FUNCTION_BLOCK Control (* Composite Function Block Type *)
  (* Standard: 61499-2 *)
  (* Version 0.0, 2/9/2018, Sandeep Patil, nxtControl GmbH, template *)
  PACKAGE Main;
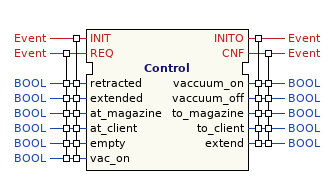
  EVENT_INPUT
    INIT WITH retracted, extended, at_magazine, at_client, empty, vac_on; (* Initialization Request *)
    REQ WITH retracted, extended, at_magazine, at_client, empty, vac_on; (* Normal Execution Request *)
  END_EVENT
  EVENT_OUTPUT
    INITO WITH vaccuum_on, vaccuum_off, to_magazine, to_client, extend; (* Initialization Confirm *)
    CNF WITH vaccuum_on, vaccuum_off, to_magazine, to_client, extend; (* Execution Confirmation *)
  END_EVENT
  VAR_INPUT
    retracted : BOOL;
    extended : BOOL;
    at_magazine : BOOL; (* Input event qualifier *)
    at_client : BOOL;
    empty : BOOL; (* Input event qualifier *)
    vac_on : BOOL;
  END_VAR
  VAR_OUTPUT
    vaccuum_on : BOOL; (* Output event qualifier *)
    vaccuum_off : BOOL;
    to_magazine : BOOL;
    to_client : BOOL;
    extend : BOOL; (* Output event qualifier *)
  END_VAR
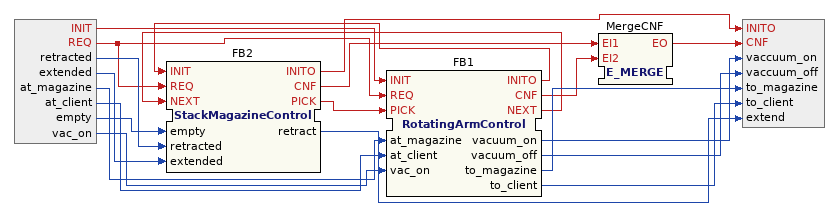
  FBS
    FB1 : RotatingArmControl;
    FB2 : StackMagazineControl;
    MergeCNF : E_MERGE;
  END_FBS
  EVENT_CONNECTIONS
    INIT TO FB1.INIT;
    REQ TO FB2.REQ;
    FB2.CNF TO MergeCNF.EI1;
    FB1.CNF TO MergeCNF.EI2;
    MergeCNF.EO TO CNF;
    REQ TO FB1.REQ;
    FB2.PICK TO FB1.PICK;
    FB1.NEXT TO FB2.NEXT;
    FB1.INITO TO FB2.INIT;
    FB2.INITO TO INITO;
  END_CONNECTIONS
  DATA_CONNECTIONS
    empty TO FB2.empty;
    retracted TO FB2.retracted;
    extended TO FB2.extended;
    at_magazine TO FB1.at_magazine;
    at_client TO FB1.at_client;
    FB1.vacuum_on TO vaccuum_on;
    FB1.vacuum_off TO vaccuum_off;
    FB1.to_magazine TO to_magazine;
    FB1.to_client TO to_client;
    FB2.retract TO extend;
    vac_on TO FB1.vac_on;
  END_CONNECTIONS
END_FUNCTION_BLOCK
